TYPE ELL18AttenuationFilterConfig EXTENDS DeviceConfiguration :
STRUCT
	SerialCommunication : SerialCommunication;
END_STRUCT
END_TYPE

(* stored: Version 1.1.0.1, ProductVersion 3.1.4024.10
   DUT ELL18AttenuationFilterConfig: Id {4c351d08-556b-4241-ad7c-bf292d79d97c} *)
